FUNCTION_BLOCK ABSTRACT FB_LinkedObject EXTENDS FB_Object IMPLEMENTS I_Object
VAR
    _ipParent:          I_LinkedObject;
END_VAR

METHOD FB_init : BOOL
VAR_INPUT
    bInitRetains:           BOOL; // if TRUE, the retain variables are initialized (warm start / cold start)
    bInCopyCode:            BOOL;  // if TRUE, the instance afterwards gets moved into the copy code (online change)
    ipParentObject:         I_LinkedObject;
END_VAR
THIS^._ipParent := ipParentObject;
END_METHOD

PROPERTY ipContext : I_Context
GET
IF THIS^._ipParent <> 0 THEN
    ipContext := THIS^.ipParent.ipContext;
END_IF
END_GET
END_PROPERTY

PROPERTY ipParent : I_LinkedObject
GET
ipParent := THIS^._ipParent;
END_GET
END_PROPERTY

END_FUNCTION_BLOCK

(* stored: Version 1.1.0.1, ProductVersion 3.1.4024.12
   POU FB_LinkedObject: Id {87ccbc5a-8a98-4cc4-aa55-78ff92f7c37f}, SpecialFunc None
   Method FB_init: Id {058b6abe-0386-4ead-9210-33fdf22e4732}
   Property ipContext: Id {af011723-3225-42bc-a3cf-ab5677defbfe}
   Get Get: Id {40949f99-26a3-42b6-8031-091b2b3252b0}
   Property ipParent: Id {476836f0-75a2-440a-a857-bf17b0a7f0dc}
   Get Get: Id {07e655a1-6465-4a2f-826a-bf0c292f7655} *)
